FUNCTION_BLOCK ABSTRACT FB_BaseAxis IMPLEMENTS I_BaseAxis
VAR_INPUT
	bEnable				: BOOL;		// enable the axis and its position control loop
	bReset				: BOOL;		// reset the axis
	bSoEReset			: BOOL;		// diagnostic reset
	bHomeAxis			: BOOL;		// Home the axis
	fPosition			: LREAL;	// position to move the axis to
	fVelocity			: LREAL;	// set the Velocity of the axis
	bMoveNeg			: BOOL;		// decrease position
	bMovePos			: BOOL;		// increase position
END_VAR
VAR_OUTPUT
	fActualPosition		: LREAL;	// actual_position of the axis
	bCalibrated			: BOOL;		// true if absolute calibration
	bError				: BOOL;		// true if error
	nErrorID			: UDINT;	// error ID of the axis
	bReady				: BOOL;		// drive is ready
END_VAR
VAR
	fbComm				: I_Comm;
	fbAxis				: FB_Axis;
	fbSoEReset			: FB_SoEReset;
	axisRef				: AXIS_REF;
END_VAR

PROPERTY ActualPosition : LREAL
GET
ActualPosition := fActualPosition;
END_GET
SET
fActualPosition := ActualPosition;
END_SET
END_PROPERTY

PROPERTY Busy : BOOL
GET
Busy := fbAxis.Busy;
END_GET
END_PROPERTY

PROPERTY Calibrated : BOOL
GET
Calibrated := bCalibrated;
END_GET
END_PROPERTY

PROPERTY Enable : BOOL
GET
Enable := bEnable;
END_GET
SET
bEnable := Enable;
END_SET
END_PROPERTY

PROPERTY Error : BOOL
GET
Error := bError;
END_GET
END_PROPERTY

PROPERTY ErrorID : UDINT
GET
ErrorID := nErrorID;
END_GET
END_PROPERTY

//FB_Init is always available implicitly and it is used primarily for initialization.
//The return value is not evaluated. For a specific influence, you can also declare the
//methods explicitly and provide additional code there with the standard initialization
//code. You can evaluate the return value.
METHOD FB_Init: BOOL
VAR_INPUT
    bInitRetains	: BOOL; // TRUE: the retain variables are initialized (reset warm / reset cold)
    bInCopyCode		: BOOL;  // TRUE: the instance will be copied to the copy code afterward (online change)
	comm			: I_Comm;   
END_VAR
THIS^.fbComm := comm;
END_METHOD

PROPERTY HomeAxis : BOOL
GET
HomeAxis := bHomeAxis;
END_GET
SET
bHomeAxis := HomeAxis;
END_SET
END_PROPERTY

PROPERTY InNegLimit : BOOL
GET
// no limit-switch input at this level; concrete subclasses must override this with a real
// hardware/soft-limit read. Left unoverridden, this always reports "not at the limit" -- the
// safe-looking value but not an accurate one (BROTLib#20)
InNegLimit := FALSE;
END_GET
END_PROPERTY

PROPERTY InPosLimit : BOOL
GET
// see InNegLimit -- same caveat, concrete subclasses must override with a real limit read
InPosLimit := FALSE;
END_GET
END_PROPERTY

PROPERTY isTracking : BOOL
GET
isTracking := fbAxis.isTracking;
END_GET
END_PROPERTY

PROPERTY MoveNeg : BOOL
GET
MoveNeg := bMoveNeg;
END_GET
SET
bMoveNeg := MoveNeg;
END_SET
END_PROPERTY

PROPERTY MovePos : BOOL
GET
MovePos := bMovePos;
END_GET
SET
bMovePos := MovePos;
END_SET
END_PROPERTY

PROPERTY Position : LREAL
GET
Position := fPosition;
END_GET
SET
fPosition := Position;
END_SET
END_PROPERTY

PROPERTY Ready : BOOL
GET
Ready := bReady;
END_GET
END_PROPERTY

METHOD Reset : BOOL
bReset := TRUE;
END_METHOD

PROPERTY Velocity : LREAL
GET
Velocity := fVelocity;
END_GET
SET
fVelocity := Velocity;
END_SET
END_PROPERTY

END_FUNCTION_BLOCK

(* stored: Version 1.1.0.1, ProductVersion 3.1.4024.15
   POU FB_BaseAxis: Id {bae85b54-65c9-4d1f-98f7-530b10d558b7}, SpecialFunc None
   Property ActualPosition: Id {119a6810-9421-4af7-8061-878d113661ac}
   Get Get: Id {4fe5f61f-7ca4-4b9a-a8e0-4b1337fe7275}
   Set Set: Id {24b1756c-cbf8-47ed-ab16-900f7081a1ba}
   Property Busy: Id {567e8af7-1006-4a9e-a236-efe3efee35b4}
   Get Get: Id {bc8cb34d-293c-40ce-ac83-5fd7efe63294}
   Property Calibrated: Id {b034059e-7dc3-4131-8628-44f1ad17bd06}
   Get Get: Id {fe3ff6d9-4050-4415-b9d6-711bddc50fae}
   Property Enable: Id {9e77bb53-50cb-4ee3-889b-4a939224a95e}
   Get Get: Id {22e8b9c7-685d-4266-b650-26373bcdabb1}
   Set Set: Id {5f0ef5ff-7479-4aad-ac7e-70298b831f6f}
   Property Error: Id {e8700151-a6f7-4979-9adf-7a637755cd40}
   Get Get: Id {918a6a55-fc48-4705-8e89-8dd3c47b45de}
   Property ErrorID: Id {a5048771-31fc-4374-9324-33f40b24b34e}
   Get Get: Id {6634ff68-5c6d-48b1-8253-67f018b99548}
   Method FB_Init: Id {c74882ff-aa80-4625-bc9f-1892a4f93fe8}
   Property HomeAxis: Id {d478184b-7b5d-4c62-b7cf-8d2b4f01dcdf}
   Get Get: Id {ba27d5dc-e1e3-47a7-9418-47220a9e0fdf}
   Set Set: Id {2f942b98-7629-4da4-99dc-e4bb1a84e0da}
   Property InNegLimit: Id {94954a80-5c0d-479c-ace0-6ef4a1491519}
   Get Get: Id {1fe9e6f2-4c2a-46e3-a448-c4853855b1c9}
   Property InPosLimit: Id {1777e73c-72ff-438e-b976-30dcfd62b989}
   Get Get: Id {d601f82d-f558-4d9f-b984-17f1ca4a9ff5}
   Property isTracking: Id {43e4a46e-8208-431f-9a95-d00464ff2604}
   Get Get: Id {064e95fd-6df9-48ee-a3f4-95fbd612c4f3}
   Property MoveNeg: Id {15f0bee2-b125-4049-9684-46d48bbd96a6}
   Get Get: Id {cafbeb19-3d1c-402f-8d01-ac78da307a6d}
   Set Set: Id {a02ef8e6-fabd-4493-83ba-b0642d198e82}
   Property MovePos: Id {215e3cb6-21ef-44de-907f-71731a297ec3}
   Get Get: Id {63d7329a-f799-4d08-ae6a-27b3a5f114b3}
   Set Set: Id {8584cc68-da28-4c0b-b3b0-bd5ca2215dae}
   Property Position: Id {5a18ed5b-37ae-4510-95dd-b35de6b1be4a}
   Get Get: Id {ada6b8a7-fcd9-46dd-a83c-0848ac5c8487}
   Set Set: Id {b6483ba5-2ead-4e18-a945-d6741047aa5c}
   Property Ready: Id {578ee6c1-3b8a-40ec-bd94-1f6e4dcf3ca3}
   Get Get: Id {4a6c02c4-b6c1-484b-9d28-b7f910e36cc3}
   Method Reset: Id {480a94e1-ff7c-412c-a535-d40e3f0b7b81}
   Property Velocity: Id {1498ec9f-a70e-40b1-bf3c-fd598252e6f2}
   Get Get: Id {566bd3aa-c6e3-4f41-889e-a7b3ad1eb487}
   Set Set: Id {a8110547-f17c-4e90-bdb3-17be6b37c36b} *)
